Fanuc KAREL source: compact_preamble.KL

PROGRAM KB00107
%NOLOCKGROUP
VAR
P1 : XYZWPREXT;RESULT:BOOLEAN
BEGIN
RESULT=IN_RANGE(P1)
END KB00107
